(* CODESYS project SPT_NC_Cam_Slave.library
   Company: Beckhoff Automation LLC
   DefaultNamespace: SPT_NCCamSlave
   Version: 3.0.0
   Placeholder: SPT NC Cam Slave
   Title: SPT NC Cam Slave

Project tree, tasks and I/O mapping:
  libraries: SPT Base Types, * (Beckhoff Automation LLC); SPT NC Axis, * (Beckhoff Automation LLC); Tc2_Math, * (Beckhoff Automation GmbH); Tc2_MC2, * (Beckhoff Automation GmbH); Tc2_MC2_Camming, * (Beckhoff Automation GmbH); Tc3_Module, * (Beckhoff Automation GmbH); Tc3_System, * (Beckhoff Automation GmbH)
  DUTs/
    data type E_CamAxisState
    data type E_CamSyncMode
    data type ST_CamParameters
    data type ST_CamPoints
  Function Blocks/
    function block FB_CamSlaveAxis [ST]: Home, MoveModulo, Reset, Stop, CamParameters, ChangeMode, FindSlavePos, FindSyncPos, InSync, Master, RunningTable, StartCouple, StartSync, SyncPos, UpdateTable, CyclicLogic, CallFBs, Initialize
  Interfaces/
    interface I_CamSlaveAxis: CamParameters, ChangeMode, FindSlavePos, FindSyncPos, InSync, Master, RunningTable, StartCouple, StartSync, SyncPos, UpdateTable
  Project Information/
    function F_GetCompany [ST]
    function F_GetTitle [ST]
    function F_GetVersion [ST]
  Version/
    global variables Global_Version
  global variables Parameters_NCCamAxis
*)

// DUTs/E_CamAxisState
{attribute 'qualified_only'}
{attribute 'strict'}
TYPE E_CamAxisState : (
        eCamAxisState_Disabled := 0,
        eCamAxisState_ReadMasterParameters,
        eCamAxisState_ReadSlaveParameters,
        eCamAxisState_AxisInitDone,
        eCamAxisState_WaitForCommand,
        eCamAxisState_DecoupleBeforeStart,
        eCamAxisState_CheckTableSelect,
        eCamAxisState_LoadCamTable,
        eCamAxisState_CheckAxisStatus,
        eCamAxisState_ReadSlaveDynamics,
        eCamAxisState_DetermineSyncMove,
        eCamAxisState_SlaveSyncMove,
        eCamAxisState_CoupleSlave,
        eCamAxisState_SetChangeMode,
        eCamAxisState_WaitForChangeCommand,
        eCamAxisState_WriteNewTable,
        eCamAxisState_WaitForActive,
        //eCamAxisState_DecoupleSlave,

        //eCamAxisState_HaltSlave,
        eCamAxisState_Error
    ) UDINT;
END_TYPE

// DUTs/E_CamSyncMode
{attribute 'qualified_only'}
{attribute 'strict'}
TYPE E_CamSyncMode : (
        eCamSyncMode_ShortestWay    := 0, // Move the Shortest Distance
        eCamSyncMode_Forward        := 1, // Move Only in the Forward Direction
        eCamSyncMode_Reverse        := 2, // Move Only in the Reverse Direction
        eCamSyncMode_Window_Forward := 3, // Move Shortest Distance If In Window Else Move Forward
        eCamSyncMode_Window_Reverse := 4  // Move Shortest Distance If In Window Else Move Reverse
    );
END_TYPE

// DUTs/ST_CamParameters
TYPE ST_CamParameters :
    STRUCT
        // Table Must Be Constructed of Motion Functions
        MasterPos    : LREAL         := 0.1;                                    // Position of Master For Which Corresponding Slave Position Is Found For
        SyncMode     : E_CamSyncMode := E_CamSyncMode.eCamSyncMode_ShortestWay; // Specifies Which Direction Slave Moves To Synchronize With the Master
        SyncWindow   : LREAL         := 10.0;                                   // Used In Conjunction With Sync Mode
        SyncVelocity : LREAL         := 10.0;                                   // Used When Slave Moves To Synchronization Position
        SyncAccel    : LREAL         := 100.0;                                  // Used When Slave Moves To Synchronization Position
        SyncDecel    : LREAL         := 100.0;                                  // Used When Slave Moves To Synchronization Position
        SyncJerk     : LREAL         := 1000.0;                                 // Used When Slave Moves To Synchronization Position

        //EmergencyDecel : LREAL         := 1000.0;                                 // Rate At Which Slave Stops On Loss of Function Block Enable or Error

        //EmergencyJerk  : LREAL         := 10000.0;                                // Rate At Which Slave Stops On Loss of Function Block Enable or Error
        TableSelect   : UDINT     := 1; // Selects Which of Five Cam Tables To Use
        CamTableId    : MC_CAM_ID := 1; // Make Sure All Your Id's are Unique
        CamTable      : ARRAY[1..Parameters_NCCamAxis.CAM_SLAVE_AXIS_TABLES] OF ST_CamPoints;
        Periodic      : BOOL         := TRUE;
        MasterOffset  : LREAL        := 0.0;
        SlaveOffset   : LREAL        := 0.0;
        MasterScaling : LREAL        := 1.0;
        SlaveScaling  : LREAL        := 1.0;
        StartMode     : MC_StartMode := MC_STARTMODE_ABSOLUTE;
        BufferMode    : MC_BufferMode;
        CamInOptions  : ST_CamInOptions;
        ChangeOptions : ST_CamInOptions; // Used for MC_SetCamOnlineChangeMode; Change Mode is Set After Cam In
    END_STRUCT
END_TYPE

// DUTs/ST_CamPoints
TYPE ST_CamPoints :
    STRUCT
        Points         : ARRAY[1..Parameters_NCCamAxis.CAM_SLAVE_AXIS_MAX_CAM_POINTS] OF MC_MotionFunctionPoint; // Array of Points 
        NumberOfPoints : DINT;                                                                                   // Quantity of Points 
    END_STRUCT
END_TYPE

// TYPE MC_MotionFunctionType

// 	MOTIONFUNCTYPE_NOTDEF,

//	MOTIONFUNCTYPE_POLYNOM1

//	MOTIONFUNCTYPE_POLYNOM3

//	MOTIONFUNCTYPE_POLYNOM5								Rest to Rest

//	MOTIONFUNCTYPE_POLYNOM8

// 	MOTIONFUNCTYPE_SINUSLINIE

//	MOTIONFUNCTYPE_MODSINUSLINIE

//	MOTIONFUNCTYPE_BESTEHORN

//	MOTIONFUNCTYPE_BESCHLTRAPEZ

//	MOTIONFUNCTYPE_POLYNOM5_MM						Motion to Motion

//	MOTIONFUNCTYPE_SINUS_GERADE_KOMBI

// 	MOTIONFUNCTYPE_HARMONIC_KOMBI_RT

//	MOTIONFUNCTYPE_HARMONIC_KOMBI_TR

//	MOTIONFUNCTYPE_HARMONIC_KOMBI_VT

//	MOTIONFUNCTYPE_HARMONIC_KOMBI_TV

//	MOTIONFUNCTYPE_BESCHLTRAPEZ_RT

//	MOTIONFUNCTYPE_BESCHLTRAPEZ_RT

//	MOTIONFUNCTYPE_MODSINUSLINIE_VV

//	MOTIONFUNCTYPE_POLYNOM7_MM

//	MOTIONFUNCTYPE_POLYNOM6STP

//	MOTIONFUNCTYPE_POLYNOM6WDP

//	MOTIONFUNCTYPE_STEPFUNCTION

// TYPE MC_MotionFunctionPoint

//	MOTIONPOINTTYPE_IGNORE

//	MOTIONPOINTTYPE_REST				Vel = 0 and Accel = 0

//	MOTIONPOINTTYPE_VELOCITY		Vel = V and Accel = 0

//	MOTIONPOINTTYPE_TURN				Vel = 0 and Accel = A

//	MOTIONPOINTTYPE_MOTION			Vel = V and Accel = A

//	MOTIONPOINTTYPE_ADD

//	MOTIONPOINTTYPE_ACTIVATION

// Version/Global_Version
{attribute 'TcGenerated'}
{attribute 'no-analysis'}
{attribute 'linkalways'}

// This function has been automatically generated from the project information.
VAR_GLOBAL CONSTANT
    {attribute 'const_non_replaced'}
    stLibVersion_SPT_NC_Cam_Slave : ST_LibVersion := (iMajor := 3, iMinor := 0, iBuild := 0, iRevision := 0, nFlags := 1, sVersion := '3.0.0');
END_VAR

// Parameters_NCCamAxis
{attribute 'qualified_only'}
VAR_GLOBAL CONSTANT
    CAM_SLAVE_AXIS_TABLES         : UDINT := 10;
    CAM_SLAVE_AXIS_MAX_CAM_POINTS : UDINT := 30;
END_VAR

// Function Blocks/FB_CamSlaveAxis
FUNCTION_BLOCK FB_CamSlaveAxis EXTENDS FB_BasicAxis IMPLEMENTS I_CamSlaveAxis
VAR
    {attribute 'hide'}
    DummyAxis                   : AXIS_REF;
    SequenceState               : UDINT;
    MCCamOut                    : MC_CamOut;
    MCCamIn                     : MC_CamIn;
    MCCamTableSelect            : MC_CamTableSelect;
    MCSetCamOnlineChangeMode    : MC_SetCamOnlineChangeMode;
    MCWriteMotionFunction       : MC_WriteMotionFunction;
    MCReadCamTableSlaveDynamics : MC_ReadCamTableSlaveDynamics;
    MasterParameters            : ST_AxisParameterSet; // Master Information 
    InWindow                    : BOOL;
    SemaphoreBusy               : BOOL;
    MoveTarget                  : LREAL;
    OldTableSelect              : UDINT;
    CurrentTableSelect          : UDINT := 1;
    CurrentPoints               : ARRAY[1..Parameters_NCCamAxis.CAM_SLAVE_AXIS_MAX_CAM_POINTS] OF MC_MotionFunctionPoint;
    CurrentTable                : MC_Cam_Ref;
    ReadSlaveDynamicsMasterPos  : LREAL;
    MoveModuloDirection         : MC_Direction;
    FindSlavePositionCommand    : BOOL; // Report Slave's Sync Position Based On Specified Master Position
    FindSyncPositionCommand     : BOOL; // Report Slave's Sync Position Based On Set Master Position 
    StartSyncCommand            : BOOL; // execute sync move if required and couple slave to master using cam table
    StartCoupleCommand          : BOOL; // couple slave to master using cam table, no sync move used
    UpdateTableCommand          : BOOL; // Update Current Cam Table
    ChangeModeCommand           : BOOL; // Update OnLineChangeMode 
    FindDone                    : BOOL; // indicates slave position lookup is complete and _SyncPos is updated
    SequenceError               : BOOL;
    SequenceErrorID             : UDINT;
    ReadyToCam                  : BOOL;
    _CamParameters              : REFERENCE TO ST_CamParameters; // Parameters for Camming Motion	
    _InSync                     : BOOL;                          // indicates slave is coupled	
    _Master                     : REFERENCE TO AXIS_REF;
    _RunningTable               : UDINT; // indicates running cam table in parameter array
    _SyncPos                    : LREAL; // indicates cam table slave position for designated master position
END_VAR

//There should be no code in the function block body

METHOD Home : BOOL
IF _Busy OR _Error OR ipHomeMethod = 0 THEN
    RETURN;
END_IF

SequenceState := 0;
Home          := SUPER^.Home();
END_METHOD

METHOD MoveModulo : BOOL
VAR_INPUT
    Position      : LREAL;
    Direction     : MC_Direction;
    AbortPrevious : BOOL;
END_VAR
IF _Error THEN
    RETURN;
ELSE
    IF (_Busy AND NOT StartSyncCommand) THEN
        RETURN;
    END_IF
END_IF

MoveModulo := SUPER^.MoveModulo(Position, Direction, AbortPrevious);
END_METHOD

METHOD Reset : BOOL
IF _Busy OR _Axis.Status.Coupled OR ipResetMethod = 0 THEN
    //If axis is coupled it should be reset through the master
    RETURN;
END_IF

IF SUPER^.Reset() THEN
    IF SequenceError THEN
        SequenceError   := FALSE;
        SequenceErrorID := 0;
        SequenceState   := E_CamAxisState.eCamAxisState_Disabled;
    END_IF

    IF MCReadCamTableSlaveDynamics.Error THEN
        MCReadCamTableSlaveDynamics(Execute := FALSE);
    END_IF

    IF __ISVALIDREF(_Master) THEN
        IF MCCamTableSelect.Error THEN
            MCCamTableSelect(Master   := _Master,
                             Slave    := _Axis,
                             CamTable := CurrentTable,
                             Execute  := FALSE);
        END_IF

        IF MCCamIn.Error THEN
            McCamIn(Master := _Master, Slave := _Axis, Execute := FALSE);
        END_IF

        IF MCCamOut.Error THEN
            McCamOut(Slave := _Axis, Execute := FALSE);
        END_IF
    END_IF

    IF MCWriteMotionFunction.Error THEN
        MCWriteMotionFunction(Execute := FALSE);
    END_IF

    IF MCSetCamOnlineChangeMode.Error THEN
        MCSetCamOnlineChangeMode(Execute := FALSE);
    END_IF

    Reset := TRUE;
END_IF
END_METHOD

METHOD Stop : BOOL
//StopCommand := TRUE;

//Stop                 := TRUE;
Stop := SUPER^.Stop();
END_METHOD

PROPERTY CamParameters : REFERENCE TO ST_CamParameters
GET
IF __ISVALIDREF(_CamParameters) THEN
    CamParameters REF= _CamParameters;
END_IF
END_GET
SET
_CamParameters REF= CamParameters;
END_SET
END_PROPERTY

METHOD ChangeMode : BOOL
VAR_INPUT
END_VAR
IF _Error OR _Busy OR NOT ReadyToCam THEN
    RETURN;
ELSE
    ChangeModeCommand := TRUE;
    ChangeMode        := TRUE;
END_IF
END_METHOD

METHOD FindSlavePos : BOOL
VAR_INPUT
END_VAR
IF _Error OR _Busy OR NOT ReadyToCam THEN
    RETURN;
ELSE
    FindSlavePositionCommand := TRUE;
    FindSlavePos             := TRUE;
END_IF
END_METHOD

METHOD FindSyncPos : BOOL
VAR_INPUT
END_VAR
IF _Error OR _Busy OR NOT ReadyToCam THEN
    RETURN;
ELSE
    FindSyncPositionCommand := TRUE;
    FindSyncPos             := TRUE;
END_IF
END_METHOD

PROPERTY InSync : BOOL
GET
InSync := _InSync;
END_GET
END_PROPERTY

PROPERTY Master : REFERENCE TO Tc2_MC2.AXIS_REF
GET
IF __ISVALIDREF(_Master) THEN
    Master REF= _Master;
END_IF
END_GET
SET
_Master REF= Master;
END_SET
END_PROPERTY

PROPERTY RunningTable : UDINT
GET
RunningTable := _RunningTable;
END_GET
END_PROPERTY

METHOD StartCouple : BOOL
VAR_INPUT
END_VAR
IF _Error OR _Busy OR NOT ReadyToCam OR NOT FindDone THEN
    RETURN;
ELSE
    StartCoupleCommand := TRUE;
    StartCouple        := TRUE;
END_IF
END_METHOD

METHOD StartSync : BOOL
VAR_INPUT
END_VAR
IF _Error OR _Busy OR NOT ReadyToCam OR _InSync THEN
    RETURN;
ELSE
    StartSyncCommand := TRUE;
    StartSync        := TRUE;
END_IF
END_METHOD

PROPERTY SyncPos : LREAL
GET
SyncPos := _SyncPos;
END_GET
END_PROPERTY

METHOD UpdateTable : BOOL
VAR_INPUT
END_VAR
IF _Error OR _Busy OR NOT ReadyToCam THEN
    RETURN;
ELSE
    UpdateTableCommand := TRUE;
    UpdateTable        := TRUE;
END_IF
END_METHOD

METHOD PUBLIC CyclicLogic
IF NOT _InitComplete THEN
    _InitComplete := THIS^.Initialize();
    RETURN;
END_IF

_InSync    := _Axis.Status.Coupled;
ReadyToCam :=
    __ISVALIDREF(_CamParameters) AND __ISVALIDREF(_Master) AND_THEN (_Master.NcToPlc.AxisId > 0) AND_THEN (_Axis.NcToPlc.AxisId > 0) AND_THEN (_Master.NcToPlc.AxisId <> _Axis.NcToPlc.AxisId);

IF _Axis.Status.Error THEN
    SequenceState := E_CamAxisState.eCamAxisState_Disabled;
END_IF

CASE SequenceState OF
    E_CamAxisState.eCamAxisState_Disabled:
        // Reset Outputs 
        SequenceError := FALSE;
        FindDone      := FALSE;
        _RunningTable := 0;
        _SyncPos      := 0.0;

        // Reset Semaphore Inputs 
        FindSlavePositionCommand := FALSE;
        FindSyncPositionCommand  := FALSE;
        StartSyncCommand         := FALSE;
        StartCoupleCommand       := FALSE;
        UpdateTableCommand       := FALSE;
        ChangeModeCommand        := FALSE;
        SequenceErrorID          := 0;

        // Reset All Function Block Calls 
        MCCamTableSelect.Execute            := FALSE;
        MCReadCamTableSlaveDynamics.Execute := FALSE;
        McCamIn.Execute                     := FALSE;
        McCamOut.Execute                    := FALSE;
        MCSetCamOnlineChangeMode.Execute    := FALSE;
        McWriteMotionFunction.Execute       := FALSE;

        // Wait for Function Block Enable 
        IF NOT _Axis.Status.Error AND ReadyToCam THEN
            // Function Block Has to Be Enabled and Slave Axis is Error Free Before Continue 
            SequenceState := E_CamAxisState.eCamAxisState_ReadMasterParameters;
        END_IF
    E_CamAxisState.eCamAxisState_ReadMasterParameters:
        MCReadParameterSet(Execute := TRUE, Parameter := MasterParameters, Axis := _Master);
        IF MCReadParameterSet.Error THEN
            //MCReadParameterSet(Execute := FALSE, Parameter := MasterParameters, Axis := _Master);
            SequenceErrorID := MCReadParameterSet.ErrorID;
            SequenceState   := E_CamAxisState.eCamAxisState_Error;
        ELSIF MCReadParameterSet.Done THEN
            MCReadParameterSet(Execute := FALSE, Parameter := MasterParameters, Axis := _Master);
            SequenceState := E_CamAxisState.eCamAxisState_AxisInitDone;
        END_IF
    E_CamAxisState.eCamAxisState_ReadSlaveParameters:
        MCReadParameterSet(Execute := TRUE, Parameter := _AxisParameters, Axis := _Axis);
        IF MCReadParameterSet.Error THEN
            //MCReadParameterSet(Execute := FALSE, Parameter := _AxisParameters, Axis := _Axis);
            SequenceErrorID := MCReadParameterSet.ErrorID;
            SequenceState   := E_CamAxisState.eCamAxisState_Error;
        ELSIF MCReadParameterSet.Done THEN
            MCReadParameterSet(Execute := FALSE, Parameter := _AxisParameters, Axis := _Axis);
            SequenceState := E_CamAxisState.eCamAxisState_AxisInitDone;
        END_IF
    E_CamAxisState.eCamAxisState_AxisInitDone:
        // Inputs Should Be Off After Initialization or After An Error 
        IF NOT FindSlavePositionCommand AND NOT FindSyncPositionCommand AND NOT StartSyncCommand AND NOT StartCoupleCommand AND NOT UpdateTableCommand THEN
            SequenceState := E_CamAxisState.eCamAxisState_WaitForCommand;
        ELSE
            SequenceState := E_CamAxisState.eCamAxisState_Error;
        END_IF
    E_CamAxisState.eCamAxisState_WaitForCommand:
        IF FindSlavePositionCommand OR FindSyncPositionCommand OR StartSyncCommand THEN
            FindDone := FALSE;

            // DeCouple Slave If Coupled 
            IF _InSync THEN
                SequenceState := E_CamAxisState.eCamAxisState_DecoupleBeforeStart;
            ELSE
                SequenceState := E_CamAxisState.eCamAxisState_CheckTableSelect;
            END_IF
        ELSIF StartCoupleCommand AND FindDone THEN
            SequenceState := E_CamAxisState.eCamAxisState_CoupleSlave;
        ELSIF ChangeModeCommand THEN
            // Can't Change Table Yet Because We Don't Have a Cam Table ID 

            // Update OnLineChangeMode 
            SequenceState := E_CamAxisState.eCamAxisState_SetChangeMode;
        END_IF
    E_CamAxisState.eCamAxisState_DecoupleBeforeStart:
        McCamOut.Execute := TRUE;
        IF NOT McCamOut.BUSY THEN
            IF McCamOut.ERROR THEN
                SequenceErrorID := McCamOut.ERRORID;
                SequenceState   := E_CamAxisState.eCamAxisState_Error;
            ELSE
                McCamOut.Execute := FALSE;
                SequenceState    := E_CamAxisState.eCamAxisState_CheckTableSelect;
            END_IF
        END_IF
    E_CamAxisState.eCamAxisState_CheckTableSelect:
        IF _CamParameters.TableSelect < 1 OR _CamParameters.TableSelect > Parameters_NCCamAxis.CAM_SLAVE_AXIS_TABLES THEN
            SequenceState := E_CamAxisState.eCamAxisState_Error;
        ELSE
            SequenceState := E_CamAxisState.eCamAxisState_LoadCamTable;
        END_IF
    E_CamAxisState.eCamAxisState_LoadCamTable:
        // Lock The Selected Table Number In Case User Changes It During Processesing 
        CurrentTableSelect := _CamParameters.TableSelect;
        CurrentPoints      := _CamParameters.CamTable[CurrentTableSelect].Points;
        OldTableSelect     := CurrentTableSelect;

        // Configure Cam Reference 
        CurrentTable.pArray      := ADR(CurrentPoints);
        CurrentTable.ArraySize   := SIZEOF(CurrentPoints);
        CurrentTable.NoOfColumns := 1; // Always 1 for Motion Functions 
        CurrentTable.NoOfRows    := DINT_TO_UDINT(_CamParameters.CamTable[CurrentTableSelect].NumberOfPoints);
        CurrentTable.TableType   := MC_TABLETYPE_MOTIONFUNCTION;
        MCCamTableSelect.Execute := TRUE;
        IF MCCamTableSelect.Error THEN
            //MCCamTableSelect.Execute := FALSE;
            SequenceErrorID := MCCamTableSelect.ErrorID;
            SequenceState   := E_CamAxisState.eCamAxisState_Error;
        ELSIF MCCamTableSelect.Done THEN
            MCCamTableSelect.Execute := FALSE;
            SequenceState            := E_CamAxisState.eCamAxisState_CheckAxisStatus;
        END_IF
    E_CamAxisState.eCamAxisState_CheckAxisStatus:
        IF _Master.Status.Error THEN
            // Master Axis Has An Error (31 = Axis Fault) 
            SequenceState := E_CamAxisState.eCamAxisState_Error;
        ELSIF NOT _Axis.Status.ControlLoopClosed THEN // 20 = Control Loop Closed 

            // Slave Axis Is Not Enabled 
            SequenceState := E_CamAxisState.eCamAxisState_Error;
        ELSIF NOT _Master.Status.ControlLoopClosed AND (MasterParameters.nAxisType = 1 OR MasterParameters.nAxisType = 3) THEN
            // Master Axis Is Not Enabled 
            SequenceState := E_CamAxisState.eCamAxisState_Error;
        ELSE
            // Find Where Slave Axis Is Suppose To Be 
            IF FindSlavePositionCommand THEN
                // Report Slave's Sync Position Based On Specified Master Position 
                ReadSlaveDynamicsMasterPos := _CamParameters.MasterPos;
                SequenceState              := E_CamAxisState.eCamAxisState_ReadSlaveDynamics;
            ELSIF FindSyncPositionCommand OR StartSyncCommand THEN
                // Report Slave's Sync Position Based On Set Master Position 
                ReadSlaveDynamicsMasterPos := _Master.NcToPlc.ActPos;
                SequenceState              := E_CamAxisState.eCamAxisState_ReadSlaveDynamics;
            ELSE
                // User Must Have Reset Inputs 
                SequenceState := E_CamAxisState.eCamAxisState_WaitForCommand;
            END_IF
        END_IF
    E_CamAxisState.eCamAxisState_ReadSlaveDynamics:
        MCReadCamTableSlaveDynamics.Execute := TRUE;
        IF MCReadCamTableSlaveDynamics.Error THEN
            //MCReadCamTableSlaveDynamics.Execute := FALSE;
            SequenceErrorID := MCReadCamTableSlaveDynamics.ErrorID;
            SequenceState   := E_CamAxisState.eCamAxisState_Error;
        ELSIF MCReadCamTableSlaveDynamics.Done THEN
            _SyncPos                            := MCReadCamTableSlaveDynamics.SlavePosition + _CamParameters.SlaveOffset;
            MCReadCamTableSlaveDynamics.Execute := FALSE;
            FindDone                            := TRUE;
            FindSlavePositionCommand            := FALSE;
            FindSyncPositionCommand             := FALSE;
            IF StartSyncCommand THEN
                SequenceState := E_CamAxisState.eCamAxisState_DetermineSyncMove;
            ELSE
                SequenceState := E_CamAxisState.eCamAxisState_WaitForCommand;
            END_IF
        END_IF
    E_CamAxisState.eCamAxisState_DetermineSyncMove:
        // If You Need to Perform a Sync Move Other Than Mode Module Then Use Inputs _FindSlave or _FindSync To Find Sync Position, Perform Move 

        // Outside of This Function Block, Then Couple Using Input _StartCouple 
        IF ABS(_Axis.NcToPlc.ModuloActPos - MODABS(MCReadCamTableSlaveDynamics.SlavePosition + _CamParameters.SlaveOffset, _AxisParameters.fEncModuloFactor)) < ABS(_CamParameters.SyncWindow) THEN
            InWindow := TRUE;
        ELSE
            InWindow := FALSE;
        END_IF

        CASE _CamParameters.SyncMode OF
            E_CamSyncMode.eCamSyncMode_ShortestWay:
                // Move the Shortest Distance 
                MoveModuloDirection := MC_Shortest_Way;
                SequenceState       := E_CamAxisState.eCamAxisState_SlaveSyncMove;
            E_CamSyncMode.eCamSyncMode_Forward:
                // Move Only in the Forward Direction 
                MoveModuloDirection := MC_Positive_Direction;
                SequenceState       := E_CamAxisState.eCamAxisState_SlaveSyncMove;
            E_CamSyncMode.eCamSyncMode_Reverse:
                // Move Only in the Reverse Direction 
                MoveModuloDirection := MC_Negative_Direction;
                SequenceState       := E_CamAxisState.eCamAxisState_SlaveSyncMove;
            E_CamSyncMode.eCamSyncMode_Window_Forward:
                // Move Shortest Distance If In Window Else Move Forward 
                IF InWindow THEN
                    MoveModuloDirection := MC_Shortest_Way;
                ELSE
                    MoveModuloDirection := MC_Positive_Direction;
                END_IF

                SequenceState := E_CamAxisState.eCamAxisState_SlaveSyncMove;
            E_CamSyncMode.eCamSyncMode_Window_Reverse:
                // Move Shortest Distance If In Window Else Move Reverse 
                IF InWindow THEN
                    MoveModuloDirection := MC_Shortest_Way;
                ELSE
                    MoveModuloDirection := MC_Negative_Direction;
                END_IF

                SequenceState := E_CamAxisState.eCamAxisState_SlaveSyncMove;
        ELSE
            SequenceState := E_CamAxisState.eCamAxisState_Error;
        END_CASE
    E_CamAxisState.eCamAxisState_SlaveSyncMove:
        Velocity     := _CamParameters.SyncVelocity;
        Acceleration := _CamParameters.SyncAccel;
        Deceleration := _CamParameters.SyncDecel;
        Jerk         := _CamParameters.SyncJerk;
        MoveTarget   := MODABS(MCReadCamTableSlaveDynamics.SlavePosition + _CamParameters.SlaveOffset, _AxisParameters.fEncModuloFactor);
        SUPER^.MoveModulo(Position := MoveTarget, Direction := MoveModuloDirection, AbortPrevious := TRUE);
        IF SUPER^.MCMoveModulo^.Error THEN
            SequenceErrorID := SUPER^.MCMoveModulo^.ErrorID;
            SequenceState   := E_CamAxisState.eCamAxisState_Error;
        ELSIF SUPER^.MCMoveModulo^.Done THEN
            SequenceState := E_CamAxisState.eCamAxisState_CoupleSlave;
        END_IF
    E_CamAxisState.eCamAxisState_CoupleSlave:
        // MC_CamIn 
        McCamIn.Execute := TRUE;
        IF McCamIn.Error THEN
            StartSyncCommand := FALSE;

            //McCamIn.Execute  := FALSE;
            SequenceErrorID := McCamIn.ErrorID;
            SequenceState   := E_CamAxisState.eCamAxisState_Error;
        ELSIF McCamIn.CommandAborted THEN
            StartSyncCommand := FALSE;
            McCamIn.Execute  := FALSE;
            SequenceState    := E_CamAxisState.eCamAxisState_Error;
        ELSIF McCamIn.InSync THEN
            // InSync May Not Report Immediately Until Slave Axis Has Past Activation Point 

            //_StartSync := FALSE;
            McCamIn.Execute := FALSE;
            _RunningTable   := CurrentTableSelect;
            SequenceState   := E_CamAxisState.eCamAxisState_SetChangeMode;
        END_IF
    E_CamAxisState.eCamAxisState_SetChangeMode:
        MCSetCamOnlineChangeMode.Execute := TRUE;
        IF MCSetCamOnlineChangeMode.Error THEN
            //MCSetCamOnlineChangeMode.Execute := FALSE;
            SequenceErrorID := MCSetCamOnlineChangeMode.ErrorID;
            SequenceState   := E_CamAxisState.eCamAxisState_Error;
        ELSIF MCSetCamOnlineChangeMode.Done THEN
            MCSetCamOnlineChangeMode.Execute := FALSE;
            ChangeModeCommand                := FALSE;
            StartSyncCommand                 := FALSE;
            StartCoupleCommand               := FALSE;
            SequenceState                    := E_CamAxisState.eCamAxisState_WaitForChangeCommand;
        END_IF
    E_CamAxisState.eCamAxisState_WaitForChangeCommand:
        IF NOT _InSync THEN
            // Axis is No Longer Coupled 
            SequenceState := E_CamAxisState.eCamAxisState_WaitForCommand;
        ELSIF ChangeModeCommand THEN
            // Update OnLineChangeMode 
            SequenceState := E_CamAxisState.eCamAxisState_SetChangeMode;
        ELSIF _CamParameters.TableSelect <> OldTableSelect OR UpdateTableCommand THEN
            // Table Number Changed or Update Current Table 
            OldTableSelect := _CamParameters.TableSelect;
            IF _CamParameters.TableSelect < 1 OR _CamParameters.TableSelect > Parameters_NCCamAxis.CAM_SLAVE_AXIS_TABLES THEN
                SequenceState := E_CamAxisState.eCamAxisState_Error;
            ELSE
                // Update Points 
                CurrentTableSelect            := _CamParameters.TableSelect;
                CurrentPoints                 := _CamParameters.CamTable[CurrentTableSelect].Points;
                CurrentTable.pArray           := ADR(CurrentPoints);
                CurrentTable.ArraySize        := SIZEOF(CurrentPoints);
                CurrentTable.NoOfColumns      := 1;
                CurrentTable.NoOfRows         := DINT_TO_UDINT(_CamParameters.CamTable[CurrentTableSelect].NumberOfPoints);
                CurrentTable.TableType        := MC_TABLETYPE_MOTIONFUNCTION;
                McWriteMotionFunction.Execute := TRUE;
                UpdateTableCommand            := TRUE;
                SequenceState                 := E_CamAxisState.eCamAxisState_WriteNewTable;
            END_IF
        END_IF
    E_CamAxisState.eCamAxisState_WriteNewTable:
        IF NOT McWriteMotionFunction.Busy THEN
            McWriteMotionFunction.Execute := FALSE;
            IF McWriteMotionFunction.Error THEN
                SequenceErrorID := McWriteMotionFunction.ErrorID;
                SequenceState   := E_CamAxisState.eCamAxisState_Error;
            ELSIF McWriteMotionFunction.Done THEN
                SequenceState := E_CamAxisState.eCamAxisState_WaitForActive;
            END_IF
        END_IF
    E_CamAxisState.eCamAxisState_WaitForActive:
        IF NOT _Axis.Status.CamDataQueued OR NOT UpdateTableCommand THEN
            // Cam Data Queued Will Not Turn Off Until Master Has Gone Past The Activation Position 

            // Abort Waiting for New Table to Activate if _UpdateTable and _UpdateTableNow Are Both Off 
            UpdateTableCommand := FALSE;
            _RunningTable      := CurrentTableSelect;
            SequenceState      := E_CamAxisState.eCamAxisState_WaitForChangeCommand;
        END_IF
    E_CamAxisState.eCamAxisState_Error: // ERROR STATE 
        FindSlavePositionCommand := FALSE;
        FindSyncPositionCommand  := FALSE;
        StartSyncCommand         := FALSE;
        StartCoupleCommand       := FALSE;
        UpdateTableCommand       := FALSE;
        ChangeModeCommand        := FALSE;

        // Wait for Reset Input
        SequenceError := TRUE;
        _Error        := TRUE;
        _ErrorID      := SequenceErrorID;
END_CASE

//Call local FBs
SUPER^.CyclicLogic();
END_METHOD

METHOD PROTECTED CallFBs : BOOL
VAR_INPUT
END_VAR
SUPER^.CallFBs();
IF __ISVALIDREF(_CamParameters) AND __ISVALIDREF(_Master) THEN
    MCReadCamTableSlaveDynamics(CamTableID := _CamParameters.CamTableId, MasterPosition := ReadSlaveDynamicsMasterPos + _CamParameters.MasterOffset);
    MCCamTableSelect(Periodic       := _CamParameters.Periodic,
                     MasterAbsolute := TRUE, // Not Implemented 
                     SlaveAbsolute  := TRUE, // Not Implemented 
                     CamTableID     := _CamParameters.CamTableId,
                     Master         := _Master,
                     Slave          := _Axis,
                     CamTable       := CurrentTable);

    McWriteMotionFunction(CamTableID := _CamParameters.CamTableId,
                          PointID    := 1,
                          NumPoints  := DINT_TO_UDINT(_CamParameters.CamTable[CurrentTableSelect].NumberOfPoints),
                          CamTable   := CurrentTable);

    MCSetCamOnlineChangeMode(ActivationMode     := _CamParameters.ChangeOptions.ActivationMode,
                             ActivationPosition := _CamParameters.ChangeOptions.ActivationPosition,
                             MasterScalingMode  := _CamParameters.ChangeOptions.MasterScalingMode,
                             SlaveScalingMode   := _CamParameters.ChangeOptions.SlaveScalingMode,
                             CamTableID         := _CamParameters.CamTableId);

    McCamIn(MasterOffset  := _CamParameters.MasterOffset,
            SlaveOffset   := _CamParameters.SlaveOffset,
            MasterScaling := _CamParameters.MasterScaling,
            SlaveScaling  := _CamParameters.SlaveScaling,
            StartMode     := _CamParameters.StartMode,
            CamTableID    := _CamParameters.CamTableId,
            BufferMode    := _CamParameters.BufferMode,
            Options       := _CamParameters.CamInOptions,
            Master        := _Master,
            Slave         := _Axis);

    McCamOut(Slave := _Axis);
END_IF

// semaphore commands on while busy
SemaphoreBusy := StartSyncCommand OR StartCoupleCommand OR FindSlavePositionCommand OR FindSyncPositionCommand OR UpdateTableCommand OR ChangeModeCommand;

//SemaphoreBusy := StartSyncCommand OR StartCoupleCommand OR StopCommand OR FindSlavePositionCommand OR FindSyncPositionCommand OR UpdateTableCommand OR ChangeModeCommand;

// ceck for function blocks busy
_Busy := _Busy OR SemaphoreBusy OR MCReadParameterSet.Busy OR MCCamTableSelect.Busy OR McCamIn.Busy OR McCamOut.Busy OR MCReadCamTableSlaveDynamics.Busy OR MCSetCamOnlineChangeMode.Busy OR
         McWriteMotionFunction.Busy;
END_METHOD

METHOD PROTECTED Initialize : BOOL
VAR_INPUT
END_VAR
IF NOT __ISVALIDREF(_Master) THEN
    _Master REF= DummyAxis;
END_IF

Initialize := SUPER^.Initialize();
END_METHOD

END_FUNCTION_BLOCK

// Interfaces/I_CamSlaveAxis
INTERFACE I_CamSlaveAxis EXTENDS I_BasicAxis

PROPERTY CamParameters : REFERENCE TO ST_CamParameters
GET
END_GET
SET
END_SET
END_PROPERTY

METHOD ChangeMode : BOOL
VAR_INPUT
END_VAR
END_METHOD

METHOD FindSlavePos : BOOL
VAR_INPUT
END_VAR
END_METHOD

METHOD FindSyncPos : BOOL
VAR_INPUT
END_VAR
END_METHOD

PROPERTY InSync : BOOL
GET
END_GET
END_PROPERTY

PROPERTY Master : REFERENCE TO AXIS_REF
GET
END_GET
SET
END_SET
END_PROPERTY

PROPERTY RunningTable : UDINT
GET
END_GET
END_PROPERTY

METHOD StartCouple : BOOL
VAR_INPUT
END_VAR
END_METHOD

METHOD StartSync : BOOL
VAR_INPUT
END_VAR
END_METHOD

PROPERTY SyncPos : LREAL
GET
END_GET
END_PROPERTY

METHOD UpdateTable : BOOL
VAR_INPUT
END_VAR
END_METHOD

END_INTERFACE

// Project Information/F_GetCompany
// This function has been automatically generated from the project information.
{attribute 'signature_flag' := '1073741824'}
{attribute 'TcGenerated'}
{attribute 'no-analysis'}
FUNCTION F_GetCompany : WSTRING
VAR_INPUT
END_VAR

F_GetCompany := "Beckhoff Automation LLC";

END_FUNCTION

// Project Information/F_GetTitle
// This function has been automatically generated from the project information.
{attribute 'signature_flag' := '1073741824'}
{attribute 'TcGenerated'}
{attribute 'no-analysis'}
FUNCTION F_GetTitle : WSTRING
VAR_INPUT
END_VAR

F_GetTitle := "SPT NC Cam Slave";

END_FUNCTION

// Project Information/F_GetVersion
// This function has been automatically generated from the project information.
{attribute 'signature_flag' := '1073741824'}
{attribute 'TcGenerated'}
{attribute 'no-analysis'}
FUNCTION F_GetVersion : ST_LibVersion
VAR_INPUT
END_VAR

F_GetVersion.iMajor    := 3;
F_GetVersion.iMinor    := 0;
F_GetVersion.iBuild    := 0;
F_GetVersion.iRevision := 0;
F_GetVersion.sVersion  := '3.0.0';
F_GetVersion.nFlags    := 1;

END_FUNCTION
